INTERFACE I_Configuration_Station

METHOD Check : BOOL
END_METHOD

METHOD PRIVATE Cmd : E_DATA_STATE
VAR_INPUT
  Ctrl      : E_DATA_CTRL;
END_VAR
END_METHOD

PROPERTY Ctrl : REFERENCE to ST_DATA_CTRL
SET
END_SET
END_PROPERTY

PROPERTY Identity : OTCID
GET
END_GET
SET
END_SET
END_PROPERTY

PROPERTY State : REFERENCE TO ST_DATA_STATE
SET
END_SET
END_PROPERTY

PROPERTY StationParameter : pointer to ARRAY[1..MAX_STATION] OF ST_STATION_PARAMETER
SET
END_SET
END_PROPERTY

END_INTERFACE

(* stored: Version 1.1.0.1
   Itf I_Configuration_Station: Id {932da42b-64b1-41d9-8b32-5909f7b3f4bd}
   Folder methods: Id {2ebf59da-ff7e-409b-9343-0809bd07dd32}
   Folder properties: Id {b17f9a43-373c-4e85-a91f-148a2346f9cf}
   Method Check: Id {b604b90c-1165-4370-ad3e-fa4e7d8f1ff7}
   Method Cmd: Id {b989bdf0-21fe-4fce-ab96-ba0f4d6ca20a}
   Property Ctrl: Id {88f69044-9534-4459-868a-f66648a23e8b}
   Set Set: Id {8ab4508d-6d12-43db-a38d-40bccf19f01b}
   Property Identity: Id {b4f69050-2b54-4909-a12a-0d56c98ccc80}
   Get Get: Id {371c1ed6-a6d6-444d-9734-4acb9113a676}
   Set Set: Id {943196ba-a396-4985-b2a2-b9d79d373b82}
   Property State: Id {74de206a-6eb0-4d3a-bd63-f029c0c1fd6a}
   Set Set: Id {336ee02a-d32c-4eb3-8752-50a55831646c}
   Property StationParameter: Id {e1e6282f-a186-4840-9550-090e98f79597}
   Set Set: Id {0faa2e24-aec0-4e14-ac0d-835ddbe55d08} *)
